PROGRAM ModeHandle
VAR
	HoldResinFlag	:	BOOL;	//Flag true after Hold Resin Condition and Until Reset
	HoldMixerFlag	:	BOOL;	//Flag true after Hold Mixer Condition and Until Reset
	StopFlag		:	BOOL;	//Flag true after Stop Condition and Until Reset
	
	testbit: BOOL;
	
END_VAR


(*Mode Handling AUTOMODE = 1 , MANUAL MODE = 2*) 
	IF GVL_HMI.ModeReqAuto =1 AND GVL_HMI.Mode = 0 AND GVL_SAF.EstopOk THEN
		GVL_HMI.Mode :=1;
		GVL_HMI.ModeReqAuto :=0;
	ELSIF GVL_HMI.ModeReqManual = 1 AND GVL_HMI.Mode = 0 AND GVL_SAF.EstopOk THEN
		GVL_HMI.Mode :=2;
		GVL_HMI.ModeReqManual := 0;
	END_IF
	
	IF GVL_HMI.ModeReqNo = 1 OR GVL_SAF.EstopOk = 0  THEN	
		GVL_HMI.Mode := 0;
		GVL_HMI.ModeReqNo := 0;
		testbit := 1;
	END_IF

	IF GVL_HMI.Mode = 0 THEN
		GVL_HMI.NoMode := 1;
		ELSE 
		GVL_HMI.NoMode := 0;
	END_IF
	IF GVL_HMI.Mode = 1 THEN
		GVL_HMI.AutoMode := 1;
		ELSE 
		GVL_HMI.AutoMode := 0;
	END_IF
	IF GVL_HMI.Mode = 2 THEN
		GVL_HMI.ManualMode := 1;
		ELSE 
		GVL_HMI.ManualMode := 0;
	END_IF
(*MCR (Master Control Reset)*)
	//Stop Conditions
	
	IF GVL_HMI.MCR = 1 THEN
	
		WX_CP.WX1(Reset_VI := 1);
		WX_CP.WX2(Reset_VI := 1);
		WX_CP.WX3(Reset_VI := 1);
		WX_CP.WX4(Reset_VI := 1);
	
		GVL_HMI.MCR			:= 0;		
		
	END_IF

END_PROGRAM

(* stored: Version 1.1.0.1, ProductVersion 3.1.4024.12
   POU ModeHandle: Id {880f8936-075f-49a8-93db-daa949b5b166}, SpecialFunc None *)
